// TIA Portal V18 export
// export: Created 2026-03-12T16:04:34.171403Z, ExportSetting WithDefaults, DisplayName Totally Integrated Automation Portal, DisplayVersion V18 Update 5, DisplayName TIA Portal Openness, DisplayVersion V18 Update 5, DisplayName TIA Portal Version Control Interface, DisplayVersion V18, DisplayName SINAMICS Startdrive Advanced, DisplayVersion V18, DisplayName SINAMICS Startdrive G130, G150, S120, S150, SINAMICS MV, S210, DisplayVersion V18, DisplayName SINAMICS Startdrive G110M, G120, G120C, G120D, G120P, G115D, DisplayVersion V18, DisplayName STEP 7 Professional, DisplayVersion V18 Update 5, DisplayName STEP 7 Safety, DisplayVersion V18, DisplayName WinCC Professional, DisplayVersion V18 Update 5
FUNCTION_BLOCK "FB WORD TO DOUBLE WORD"   // FB26, SCL
{ S7_Optimized_Access := 'TRUE' }
VERSION : 0.1
// stored: AutoNumber true, IsIECCheckEnabled false, IsRetainMemResEnabled false, MemoryReserve 100, SetENOAutomatically false, UDAEnableTagReadback false
   VAR_INPUT
      SIGNAL_Word0 : Word;   // Sinal de entrada 1
      SIGNAL_Word1 : Word;   // Sinal de entrada 2
      SIGNAL_Word2 : Word;
      SIGNAL_Word3 : Word;
      SIGNAL_Word4 : Word;
      SIGNAL_Word5 : Word;
      SIGNAL_Word6 : Word;
      SIGNAL_Word7 : Word;
      SIGNAL_Word8 : Word;
      SIGNAL_Word9 : Word;
      SIGNAL_Word10 : Word;
      SIGNAL_Word11 : Word;
      SIGNAL_Word12 : Word;
      SIGNAL_Word13 : Word;
      SIGNAL_Word14 : Word;
      SIGNAL_Word15 : Word;
   END_VAR
   VAR_OUTPUT
      BITS_TO_DWORD_0 : DWord;   // Word de saída com os sinais montados
      BITS_TO_DWORD_1 : DWord;
      BITS_TO_DWORD_2 : DWord;
      BITS_TO_DWORD_3 : DWord;
      BITS_TO_DWORD_4 : DWord;
      BITS_TO_DWORD_5 : DWord;
      BITS_TO_DWORD_6 : DWord;
      BITS_TO_DWORD_7 : DWord;
   END_VAR
BEGIN
   // Word Alarmes - Montando WORD'S em uma double word

   // Bits recebidos de campo
   #BITS_TO_DWORD_0 := (SHL(IN := WORD_TO_DWORD(#SIGNAL_Word1), N := 16) OR (#SIGNAL_Word0));
   #BITS_TO_DWORD_1 := (SHL(IN := WORD_TO_DWORD(#SIGNAL_Word3), N := 16) OR (#SIGNAL_Word2));
   #BITS_TO_DWORD_2 := (SHL(IN := WORD_TO_DWORD(#SIGNAL_Word5), N := 16) OR (#SIGNAL_Word4));
   #BITS_TO_DWORD_3 := (SHL(IN := WORD_TO_DWORD(#SIGNAL_Word7), N := 16) OR (#SIGNAL_Word6));
   #BITS_TO_DWORD_4 := (SHL(IN := WORD_TO_DWORD(#SIGNAL_Word9), N := 16) OR (#SIGNAL_Word8));
   #BITS_TO_DWORD_5 := (SHL(IN := WORD_TO_DWORD(#SIGNAL_Word11), N := 16) OR (#SIGNAL_Word10));
   #BITS_TO_DWORD_6 := (SHL(IN := WORD_TO_DWORD(#SIGNAL_Word13), N := 16) OR (#SIGNAL_Word12));
   #BITS_TO_DWORD_7 := (SHL(IN := WORD_TO_DWORD(#SIGNAL_Word15), N := 16) OR (#SIGNAL_Word14));
END_FUNCTION_BLOCK
